(* IEC 61131-3 sources: library-inventory-agv/src/communication, 2 files *)

(* ---- NavigationApiClient.st ---- *)
// =============================================================================
// NavigationApiClient — HTTP REST Client for Navigation System
// =============================================================================
// Implements the PLC-side HTTP client that communicates with the external
// navigation system at 192.168.3.100:7000.
//
// Uses CODESYS Web Client SL and JSON Utilities SL libraries to construct
// JSON request bodies and parse responses.
//
// Endpoints implemented:
//   POST /api/template/navigating      — Submit navigation task
//   POST /api/template/confirm         — Confirm task template
//   POST /api/navigating/stop          — Abort navigation
//   POST /api/navigating/charging_station/docking   — Dock at charger
//   POST /api/navigating/charging_station/undocking  — Leave charger
//   POST /api/charging/start           — Begin charging
//   POST /api/charging/stop            — End charging
//   POST /api/docking/cancel           — Cancel docking
//   GET  /api/ws                       — WebSocket status (handled separately)
// =============================================================================

FUNCTION_BLOCK NavigationApiClient
VAR_INPUT
    bExecute        : BOOL;             // Rising edge triggers request
    sEndpoint       : STRING(255);      // API path (e.g., '/api/template/navigating')
    sMethod         : STRING(10);       // 'POST' or 'GET'

    // Optional JSON body fields
    sTaskNumber     : STRING(80);       // Task identifier
    sPointName      : STRING(80);       // Waypoint name
    rDockX          : REAL;             // Docking X coordinate
    rDockY          : REAL;             // Docking Y coordinate
    rDockA          : REAL;             // Docking angle
    bIncludeCoords  : BOOL;             // Include x/y/a in JSON body
END_VAR

VAR_OUTPUT
    bDone           : BOOL;             // Request completed successfully
    bBusy           : BOOL;             // Request in progress
    bError          : BOOL;             // Request failed
    nHttpStatus     : INT;              // HTTP response status code
    sResponse       : STRING(1000);     // Response body
END_VAR

VAR
    // CODESYS Web Client SL
    fbHttpClient    : WebClient.HTTPClient;
    fbRequest       : WebClient.HTTPRequest;

    // JSON construction (JSON Utilities SL)
    pJsonData       : POINTER TO JSON.JSONData;
    factory         : JSON.JSONDataFactory;
    fbJBuilder      : JSON.fb_JBuilder;
    jsonWriter      : JSON.JSONByteArrayWriter;
    wsJsonData      : WSTRING(1000);    // JSON output buffer

    // Internal state
    eReqState       : INT;              // 0=idle, 1=building, 2=sending, 3=waiting, 4=done
    rtExecute       : R_TRIG;
    diRootIndex     : DINT;

    // Configuration
    C_BASE_URL      : STRING(80) := 'http://192.168.3.100:7000';
    C_CONTENT_TYPE  : STRING(40) := 'Content-Type: application/json';
    C_TIMEOUT       : TIME := T#5S;
    tTimeout        : TON;
END_VAR

// =========================================================================
// Execution Logic
// =========================================================================
rtExecute(CLK := bExecute);

CASE eReqState OF

0: // IDLE
    bDone := FALSE;
    bBusy := FALSE;
    bError := FALSE;

    IF rtExecute.Q THEN
        bBusy := TRUE;
        eReqState := 1;
    END_IF

1: // BUILD JSON BODY
    // Create JSON document
    pJsonData := factory.Create();
    fbJBuilder(pJsonData := pJsonData, diRootObj => diRootIndex);

    // Add task_number if provided
    IF LEN(sTaskNumber) > 0 THEN
        JSON.JsonObjectAddString(
            pJsonData   := pJsonData,
            diObject    := diRootIndex,
            wsKey       := "task_number",
            wsValue     := STRING_TO_WSTRING(sTaskNumber)
        );
    END_IF

    // Add point name if provided
    IF LEN(sPointName) > 0 THEN
        JSON.JsonObjectAddString(
            pJsonData   := pJsonData,
            diObject    := diRootIndex,
            wsKey       := "point",
            wsValue     := STRING_TO_WSTRING(sPointName)
        );
    END_IF

    // Add docking coordinates if needed
    IF bIncludeCoords THEN
        JSON.JsonObjectAddNumber(
            pJsonData   := pJsonData,
            diObject    := diRootIndex,
            wsKey       := "x",
            lrValue     := REAL_TO_LREAL(rDockX)
        );
        JSON.JsonObjectAddNumber(
            pJsonData   := pJsonData,
            diObject    := diRootIndex,
            wsKey       := "y",
            lrValue     := REAL_TO_LREAL(rDockY)
        );
        JSON.JsonObjectAddNumber(
            pJsonData   := pJsonData,
            diObject    := diRootIndex,
            wsKey       := "a",
            lrValue     := REAL_TO_LREAL(rDockA)
        );
    END_IF

    // Serialize to string
    jsonWriter(
        xExecute    := TRUE,
        pwData      := ADR(wsJsonData),
        udiSize     := SIZEOF(wsJsonData),
        jsonData    := pJsonData^,
        xAsyncMode  := FALSE
    );

    eReqState := 2;

2: // SEND HTTP REQUEST
    fbRequest(
        sUrl            := CONCAT(C_BASE_URL, sEndpoint),
        sMethod         := sMethod,
        sContentType    := 'application/json',
        sBody           := WSTRING_TO_STRING(wsJsonData),
        tTimeout        := C_TIMEOUT
    );

    fbHttpClient.SendRequest(pRequest := ADR(fbRequest));
    tTimeout(IN := TRUE, PT := C_TIMEOUT);
    eReqState := 3;

3: // WAIT FOR RESPONSE
    IF fbHttpClient.xDone THEN
        nHttpStatus := fbHttpClient.iStatusCode;
        sResponse   := fbHttpClient.sResponseBody;
        tTimeout(IN := FALSE);

        IF nHttpStatus >= 200 AND nHttpStatus < 300 THEN
            bDone := TRUE;
        ELSE
            bError := TRUE;
        END_IF

        // Clean up JSON data
        factory.Delete(pJsonData);
        bBusy := FALSE;
        eReqState := 0;

    ELSIF tTimeout.Q THEN
        tTimeout(IN := FALSE);
        factory.Delete(pJsonData);
        bError := TRUE;
        bBusy := FALSE;
        eReqState := 0;
    END_IF

END_CASE

(* ---- SensorTcpClient.st ---- *)
// =============================================================================
// SensorTcpClient — TCP Socket Client for RFID & Vision Sensors
// =============================================================================
// Manages TCP connections to the RFID reader and vision camera.
// Provides request/response pattern with timeout and reconnection logic.
//
// The RFID reader and vision camera communicate via raw TCP:
//   1. PLC sends a trigger command (scan request)
//   2. Device performs operation (RFID read / image capture + OCR)
//   3. Device returns result data
//   4. PLC parses result and updates inventory count
//
// Connection monitoring:
//   HMI_RFID_ConnectionActive   — RFID reader TCP alive
//   HMI_Vision_ConnectionActive — Vision camera TCP alive
// =============================================================================

FUNCTION_BLOCK SensorTcpClient
VAR_INPUT
    sServerIP       : STRING(15);       // Device IP address
    uiServerPort    : UINT;             // Device TCP port
    bConnect        : BOOL;             // Enable connection
    bSendRequest    : BOOL;             // Trigger data request
    sSendData       : STRING(255);      // Request payload
END_VAR

VAR_OUTPUT
    bConnected      : BOOL;             // TCP connection established
    bDataReady      : BOOL;             // Response received
    bError          : BOOL;             // Communication error
    sRecvData       : STRING(2000);     // Received response data
    nItemCount      : INT;              // Parsed: number of items detected
    nErrorCode      : DWORD;            // TCP error code
END_VAR

VAR
    // CODESYS TCP library function blocks
    fbClient        : NBS.TCP_Client;
    fbRead          : NBS.TCP_Read;
    fbWrite         : NBS.TCP_Write;

    // Connection management
    eConnState      : INT;              // 0=disconnected, 1=connecting, 2=connected
    tReconnect      : TON;              // Reconnection delay timer
    nReconnectCount : INT;              // Reconnection attempt counter

    // Request/Response state
    eReqState       : INT;              // 0=idle, 1=sending, 2=waiting, 3=done
    rtSendReq       : R_TRIG;
    tRespTimeout    : TON;

    // Buffers
    abyRecvBuffer   : ARRAY[0..2047] OF BYTE;
    uiBytesRecv     : UINT;

    // Constants
    C_RECONNECT_DELAY : TIME := T#3S;
    C_RESP_TIMEOUT    : TIME := T#5S;
    C_MAX_RECONNECT   : INT  := 5;
END_VAR

// =========================================================================
// Connection Management
// =========================================================================
CASE eConnState OF

0: // DISCONNECTED
    bConnected := FALSE;
    IF bConnect THEN
        fbClient(
            xEnable     := TRUE,
            sAddr       := sServerIP,
            uiPort      := uiServerPort
        );
        eConnState := 1;
    END_IF

1: // CONNECTING
    fbClient(xEnable := TRUE);

    IF fbClient.xActive THEN
        eConnState := 2;
        bConnected := TRUE;
        nReconnectCount := 0;
    ELSIF fbClient.xError THEN
        fbClient(xEnable := FALSE);
        nReconnectCount := nReconnectCount + 1;

        IF nReconnectCount < C_MAX_RECONNECT THEN
            tReconnect(IN := TRUE, PT := C_RECONNECT_DELAY);
            IF tReconnect.Q THEN
                tReconnect(IN := FALSE);
                eConnState := 0;    // Retry
            END_IF
        ELSE
            bError := TRUE;         // Give up after max retries
        END_IF
    END_IF

2: // CONNECTED
    bConnected := TRUE;

    // Monitor connection health
    IF NOT fbClient.xActive THEN
        bConnected := FALSE;
        eConnState := 0;           // Connection lost, auto-reconnect
    END_IF

END_CASE

// =========================================================================
// Request / Response Handling
// =========================================================================
rtSendReq(CLK := bSendRequest);

CASE eReqState OF

0: // IDLE
    bDataReady := FALSE;

    IF rtSendReq.Q AND bConnected THEN
        eReqState := 1;
    END_IF

1: // SENDING REQUEST
    fbWrite(
        xExecute    := TRUE,
        hConnection := fbClient.hConnection,
        pData       := ADR(sSendData),
        udiSize     := INT_TO_UDINT(LEN(sSendData))
    );

    IF fbWrite.xDone THEN
        fbWrite(xExecute := FALSE);
        tRespTimeout(IN := TRUE, PT := C_RESP_TIMEOUT);
        eReqState := 2;
    ELSIF fbWrite.xError THEN
        fbWrite(xExecute := FALSE);
        bError := TRUE;
        eReqState := 0;
    END_IF

2: // WAITING FOR RESPONSE
    fbRead(
        xEnable     := TRUE,
        hConnection := fbClient.hConnection,
        pData       := ADR(abyRecvBuffer),
        udiSize     := SIZEOF(abyRecvBuffer)
    );

    IF fbRead.udiCount > 0 THEN
        // Data received
        fbRead(xEnable := FALSE);
        tRespTimeout(IN := FALSE);

        uiBytesRecv := UDINT_TO_UINT(fbRead.udiCount);
        // Copy to output string (simplified — real impl handles encoding)
        MEMUtils.MemCpy(
            pDest := ADR(sRecvData),
            pSrc  := ADR(abyRecvBuffer),
            udiCount := MIN(fbRead.udiCount, SIZEOF(sRecvData) - 1)
        );

        // Parse item count from response
        // (actual parsing depends on device protocol — simplified here)
        nItemCount := ParseItemCount(sRecvData);

        bDataReady := TRUE;
        eReqState := 0;

    ELSIF tRespTimeout.Q THEN
        // Timeout — no response from sensor
        fbRead(xEnable := FALSE);
        tRespTimeout(IN := FALSE);
        bError := TRUE;
        nItemCount := 0;
        eReqState := 0;
    END_IF

END_CASE

// =========================================================================
// Disconnect handling
// =========================================================================
IF NOT bConnect THEN
    fbClient(xEnable := FALSE);
    bConnected := FALSE;
    eConnState := 0;
    eReqState := 0;
END_IF
